Yaskawa INFORM job: SKRZYNIA_5540_0_STOPNI_1OBR.JBI

/JOB
//NAME SKRZYNIA_5540_0_STOPNI_1OBR
///FOLDERNAME 02-SKRZYNIE_JOBS
//POS
///NPOS 539,539,0,45,0,0
///TOOL 0
///POSTYPE PULSE
///PULSE
C00000=1055,-24125,84372,288,19725,204
C00001=1055,-24125,84372,288,19725,204
C00002=0,-15438,65714,0,-68532,0
C00003=25524,-25821,36823,19654,-58495,38520
C00004=25524,-25821,36823,19654,-58495,38520
C00005=23988,-24960,37134,18595,-57837,38812
C00006=22822,-23954,37534,17811,-57199,39017
C00007=22935,-24057,37491,17887,-57262,38997
C00008=20006,-24258,37408,15644,-56932,39751
C00009=24402,-25289,37013,18874,-58060,38740
C00010=22585,-24665,40358,17164,-59622,30036
C00011=23477,-23257,40205,18030,-58646,29630
C00012=22519,-22398,40568,17384,-58125,29795
C00013=22700,-22567,40495,17506,-58225,29764
C00014=19339,-22794,40398,14955,-57865,30607
C00015=24825,-24328,39798,18931,-59350,29401
C00016=25524,-25821,36823,19654,-58495,38520
C00017=23988,-24960,37134,18595,-57837,38812
C00018=22822,-23954,37534,17811,-57199,39017
C00019=22935,-24057,37491,17887,-57262,38997
C00020=20006,-24258,37408,15644,-56932,39751
C00021=24402,-25289,37013,18874,-58060,38740
C00022=22585,-24665,40358,17164,-59622,30036
C00023=23477,-23257,40205,18030,-58646,29630
C00024=22519,-22398,40568,17384,-58125,29795
C00025=22700,-22567,40495,17506,-58225,29764
C00026=19339,-22794,40398,14955,-57865,30607
C00027=24825,-24328,39798,18931,-59350,29401
C00028=32755,-32613,25711,29640,-48730,33694
C00029=25632,-30899,26166,23992,-46203,35378
C00030=24264,-29862,26497,22996,-45413,35639
C00031=24403,-29974,26459,23097,-45496,35612
C00032=20575,-30233,26374,19602,-44891,36810
C00033=26556,-31526,25988,24663,-46720,35206
C00034=30846,-32795,25752,28021,-48338,30427
C00035=24953,-30697,26306,23444,-45946,31743
C00036=23937,-29910,26558,22702,-45353,31936
C00037=24039,-29993,26530,22778,-45414,31916
C00038=20322,-30240,26449,19379,-44834,33080
C00039=25997,-31433,26093,24205,-46535,31545
C00040=26028,-43665,26580,-39946,8682,24640
C00041=27956,-30595,53065,-101898,6609,54413
C00042=26028,-43663,26580,-39944,8677,24639
C00043=38124,-35330,25507,26155,-45940,34419
C00044=17528,-33021,25719,14295,-44761,40001
C00045=28412,-21339,35361,20830,-70681,36412
C00046=27333,-20260,35973,20228,-70115,36596
C00047=27560,-20497,35837,20355,-70235,36556
C00048=24830,-20816,35654,18694,-69859,37222
C00049=28877,-18893,40191,20941,-72149,36569
C00050=27817,-32566,25782,25532,-47502,36865
C00051=25779,-31294,26110,24054,-46400,37243
C00052=24344,-30243,26427,23007,-45578,37515
C00053=24432,-30312,26405,23072,-45630,37498
C00054=20021,-30599,26315,19050,-44944,38872
C00055=26262,-31616,26021,24405,-46667,37153
C00056=27439,-32346,25835,25259,-47302,36935
C00057=26020,-31415,26075,24237,-46513,37193
C00058=24581,-30384,26384,23190,-45695,37464
C00059=24689,-30466,26358,23269,-45758,37444
C00060=20001,-30771,26264,18999,-45026,38899
C00061=26308,-31607,26026,24448,-46671,37139
C00062=27526,-32360,25834,25329,-47326,36914
C00063=24645,-40364,6410,30045,-34429,34156
C00064=22958,-37632,10123,27061,-35370,35326
C00065=22703,-41294,1722,31272,-29953,33282
C00066=19440,-41515,1663,27208,-29122,34832
C00067=25465,-43501,1200,33269,-31905,32752
C00068=54276,-43673,-470,62120,-47739,23626
C00069=54276,-43673,-470,62120,-47739,23626
C00070=41752,-40945,238,55421,-40682,25053
C00071=39867,-39951,547,54583,-39468,25162
C00072=39963,-40004,529,54625,-39531,25157
C00073=37168,-40414,400,52318,-38319,25966
C00074=43368,-42081,-2849,57747,-40820,23950
C00075=4794,-34097,38974,4189,-31824,-1302
C00076=4794,-34097,38974,4189,13412,-1302
C00077=11237,-37131,38982,-12694,5333,8253
///LIMIT ON
C00078=18252,-32243,53492,22663,-13662,-6677
///LIMIT OFF
C00079=13219,-33034,38361,14494,-24384,-4511
C00080=38095,-40136,7813,41252,-44156,24924
C00081=33231,-38681,8176,37792,-41757,25918
C00082=31538,-37640,8473,36716,-40716,26179
C00083=31687,-37737,8444,36811,-40809,26155
C00084=27389,-38154,8322,32773,-39589,27627
C00085=33834,-39023,8084,38175,-42120,25821
C00086=9520,-44470,15692,8941,-38846,5030
C00087=4264,-34194,25387,4006,-26954,-81856
C00088=17634,-23800,39238,9573,-31425,-73339
C00089=17634,-23800,39238,9573,-31425,-73339
C00090=16549,-22464,39800,8390,-30730,-72975
C00091=16684,-22641,39722,8536,-30818,-73021
C00092=16684,-19968,45512,8078,-32771,-72767
C00093=17634,-23800,39238,9573,-31425,-73339
C00094=17837,-21535,44509,9322,-33342,-73155
C00095=17837,-21535,44509,9322,-33342,-73155
C00096=16866,-20378,45014,8305,-32755,-72853
C00097=17032,-20588,44918,8481,-32857,-72905
C00098=17032,-17542,51480,8009,-35060,-72636
C00099=17837,-21535,44509,9322,-33342,-73155
C00100=-20829,-18800,50532,-12466,-37179,-77446
C00101=-19934,-17904,50946,-11618,-36715,-77676
C00102=-20044,-18019,50891,-11723,-36773,-77647
C00103=-20044,-15288,56753,-11218,-38713,-77950
C00104=-20966,-18928,50473,-12596,-37250,-77413
C00105=-20884,-26676,33664,-14451,-31668,-76336
C00106=-20884,-26676,33664,-14451,-31668,-76336
C00107=-19557,-25338,34176,-13080,-30873,-76751
C00108=-19691,-25483,34117,-13220,-30955,-76709
C00109=-19691,-22773,39998,-12506,-32911,-77106
C00110=-20642,-26447,33747,-14206,-31526,-76411
C00111=-33629,-40566,17444,-29603,-33447,-71192
C00112=-33629,-40566,17444,42578,-32312,-84654
C00113=-42160,-31266,16400,42578,-32312,-84654
C00114=-87798,-804,48829,-20188,-26072,-60966
C00115=-76454,-11934,10236,-25964,7954,-64922
C00116=-76448,-11928,10235,-25961,7944,-64914
C00117=-68643,-7759,-23318,-14097,50582,-74897
C00118=-70868,-8793,-8075,-29663,30364,-70765
C00119=-67243,-1968,12282,-49553,26687,-63567
C00120=-68655,-309,14069,-48513,25966,-64203
C00121=-67497,-1678,12591,-49367,26558,-63682
C00122=-71436,-723,2905,-26484,35140,-73726
C00123=-71436,176,6426,-27636,33595,-73066
C00124=-71434,778,8668,-28412,32633,-72624
C00125=-68624,-2689,-85,-28291,36551,-72622
C00126=-99375,3692,5712,40719,48607,-84097
C00127=-94964,4957,10918,40408,44640,-83792
C00128=-93063,6047,12199,39572,43744,-83178
C00129=-94964,4957,10918,40408,44640,-83792
C00130=-94964,5754,13918,41385,43553,-84439
C00131=-94964,4957,10918,40408,44640,-83792
C00132=-90271,-412,-5146,23417,46876,-76529
C00133=-83133,-4088,-8267,6704,41492,-71542
C00134=-83133,-4088,-8267,6704,41492,-71542
C00135=-83133,-4088,-8267,6704,41492,-11598
C00136=-83133,-16026,-8267,6704,41492,-11598
C00137=-83133,-16026,-8267,6704,41492,-11598
C00138=-48225,-19387,30619,3889,32460,-6728
C00139=56943,-39861,25115,1795,-37402,-69601
C00140=29960,-38386,-19607,-115769,-41858,-24264
C00141=65721,-6478,18155,-133323,-22195,3361
C00142=70544,4411,32968,-134868,-18623,4660
C00143=71874,8263,38598,-134556,-17327,4659
C00144=72629,9390,40002,-135279,-16924,5107
C00145=71441,7638,37831,-134139,-17555,4406
C00146=77146,8888,25050,-166574,-32612,18372
C00147=77146,10029,28643,-166204,-31014,18167
C00148=77146,11198,32202,-165803,-29459,17947
C00149=75508,4678,16951,-165715,-35157,17778
C00150=68680,12216,24468,-164340,-40455,-13359
C00151=68362,12845,25743,-164045,-40097,-13561
C00152=68362,13700,28585,-163752,-38808,-13742
C00153=68362,12845,25743,-164045,-40097,-13561
C00154=64993,-1168,28876,-102971,-10760,-49875
C00155=63888,481,30670,-102324,-11438,-50313
C00156=64993,-1168,28876,-102971,-10760,-49875
C00157=58588,-14653,4620,-120782,-19611,-35794
C00158=29960,-38386,-19607,-115769,-41858,-24264
C00159=56943,-39861,25115,1795,-37402,-69601
C00160=-1002,-39861,25115,1795,-37402,-69601
C00161=-1001,-39858,25114,1795,-37402,0
///LIMIT ON
C00162=6591,-33902,35532,5956,-1761,-1932
///LIMIT OFF
C00163=6592,-33900,35531,103508,-35512,-26314
C00164=-99253,-13690,44082,59847,13407,-31313
C00165=-85045,-36869,-4353,28502,-22832,-52282
C00166=-92346,-18713,13565,21110,-22545,-55257
C00167=-85370,-14218,16934,32905,-23649,-60330
C00168=-84150,-13282,17685,34842,-23935,-61163
C00169=-82877,-12536,18624,36445,-24482,-61818
C00170=-84150,-13282,17685,34842,-23935,-61163
C00171=-85467,-11480,19558,33086,-23405,-60436
C00172=-84150,-13282,17685,34842,-23935,-61163
C00173=-85732,-21202,11427,30682,-24763,-59235
C00174=-84559,-15616,15722,33768,-24118,-60665
C00175=-84150,-13282,17685,34842,-23935,-61163
C00176=-83260,-12880,18034,36130,-24218,-61709
C00177=-84150,-13282,17685,34842,-23935,-61163
C00178=-85365,-11775,19006,33430,-23307,-60600
C00179=-84150,-13282,17685,34842,-23935,-61163
C00180=-85786,-16909,14677,31743,-23900,-59790
C00181=-84150,-13282,17685,34842,-23935,-61163
C00182=-83215,-12861,18051,36194,-24233,-61735
C00183=-84150,-13282,17685,34842,-23935,-61163
C00184=-85327,-11825,18959,33476,-23327,-60618
C00185=-84150,-13282,17685,34842,-23935,-61163
C00186=-87841,-18519,13420,28367,-23534,-58339
C00187=-84150,-13282,17685,34842,-23935,-61163
C00188=-83292,-12894,18020,36083,-24208,-61688
C00189=-84150,-13282,17685,34842,-23935,-61163
C00190=-85185,-12008,18799,33646,-23400,-60687
C00191=-84150,-13282,17685,34842,-23935,-61163
C00192=-86371,-18277,13606,30568,-23951,-59265
C00193=-84345,-13370,17612,34554,-23873,-61041
C00194=-83240,-12871,18042,36158,-24225,-61720
C00195=-84345,-13370,17612,34554,-23873,-61041
C00196=-85365,-12110,18711,33368,-23345,-60568
C00197=-84345,-13370,17612,34554,-23873,-61041
C00198=-86191,-19647,12567,30467,-24278,-59187
C00199=-84345,-13372,17610,34552,-23873,-61039
C00200=-83096,-12807,18098,36363,-24268,-61804
C00201=-84345,-13372,17610,34552,-23873,-61039
C00202=-85268,-12232,18600,33480,-23393,-60612
C00203=-84345,-13372,17610,34552,-23873,-61039
C00204=-84814,-16043,15376,33312,-24093,-60464
C00205=-84104,-13265,17702,34906,-23948,-61189
C00206=-82960,-12743,18153,36555,-24313,-61887
C00207=-84104,-13265,17702,34906,-23948,-61189
C00208=-84979,-12194,18635,33901,-23496,-60788
C00209=-84104,-13265,17702,34906,-23948,-61189
C00210=-86610,-16845,14732,30573,-23614,-59301
C00211=-84104,-13265,17702,34906,-23948,-61189
C00212=-82793,-12667,18222,36790,-24370,-61986
C00213=-84104,-13265,17702,34906,-23948,-61189
C00214=-84888,-12305,18537,34004,-23540,-60830
C00215=-84104,-13265,17702,34906,-23948,-61189
C00216=-83806,-19585,12613,33764,-25080,-60559
C00217=-83675,-13072,17868,35530,-24083,-61453
C00218=-82553,-12556,18319,37130,-24451,-62127
C00219=-83675,-13072,17868,35530,-24083,-61453
C00220=-84378,-12223,18610,34735,-23716,-61138
C00221=-83675,-13072,17868,35530,-24083,-61453
C00222=-87149,-17993,13826,29513,-23647,-58830
C00223=-84104,-13265,17702,34906,-23948,-61189
C00224=-82640,-12594,18285,37014,-24425,-62079
C00225=-84104,-13265,17702,34906,-23948,-61189
C00226=-84792,-12429,18430,34119,-23592,-60877
C00227=-84104,-13265,17702,34906,-23948,-61189
C00228=-83583,-9185,30892,23668,-36042,-57025
C00229=-85789,-8328,35795,20592,-37093,-55378
C00230=-85786,-16735,14816,31782,-23869,-59812
C00231=-84103,-13263,17702,34906,-23947,-61191
C00232=-83225,-12865,18046,36177,-24227,-61729
C00233=-84103,-13263,17702,34906,-23947,-61191
C00234=-84774,-12447,18412,34138,-23599,-60886
C00235=-84103,-13263,17702,34906,-23947,-61191
C00236=-86149,-16246,6730,18897,-35239,-57128
C00237=-86244,-15289,7532,18875,-35060,-57127
C00238=-85361,-14893,7870,19824,-35193,-57574
C00239=-86244,-15289,7532,18875,-35060,-57127
C00240=-86889,-14409,8282,18264,-34784,-56850
C00241=-86244,-15289,7532,18875,-35060,-57127
C00242=-90262,-21765,2389,14114,-35574,-54847
C00243=-90262,-21765,2389,28730,-17672,-54847
C00244=-89967,-19086,25635,28730,-17672,-54847
C00245=568,-24029,84339,168,19981,112
C00246=568,-24677,83015,164,20405,113
C00247=101153,-24598,83176,165,20353,113
C00248=101153,-24598,83176,165,20353,113
C00249=89967,-19086,25635,-28730,-17672,54847
C00250=90262,-21765,2389,-28730,-17672,54847
C00251=86932,-18662,4771,-17876,-35519,56628
C00252=86578,-15436,7408,-18515,-35011,56957
C00253=85428,-14922,7844,-19753,-35183,57541
C00254=84405,-14447,8250,-20842,-35348,58054
C00255=85428,-14922,7844,-19753,-35183,57541
C00256=86134,-13973,8661,-19091,-34881,57237
C00257=85428,-14922,7844,-19753,-35183,57541
C00258=85786,-16735,14816,-31782,-23869,59812
C00259=83514,-12996,17929,-35760,-24132,61552
C00260=82296,-12429,18424,-37488,-24534,62281
C00261=83514,-12996,17929,-35760,-24132,61552
C00262=84266,-12085,18725,-34910,-23738,61214
C00263=83514,-12996,17929,-35760,-24132,61552
C00264=87323,-6914,39851,-18853,-38149,44508
C00265=83118,-12818,18089,-36330,-24263,61791
C00266=81969,-12276,18566,-37944,-24648,62472
C00267=83118,-12818,18089,-36330,-24263,61791
C00268=83927,-11846,18941,-35423,-23842,61433
C00269=83118,-12818,18089,-36330,-24263,61791
C00270=83806,-19585,12613,-33764,-25080,60559
C00271=83148,-12832,18077,-36287,-24254,61773
C00272=81889,-12236,18598,-38058,-24676,62520
C00273=83148,-12832,18077,-36287,-24254,61773
C00274=83900,-11930,18867,-35446,-23862,61440
C00275=83148,-12832,18077,-36287,-24254,61773
C00276=86610,-16845,14732,-30573,-23614,59301
C00277=82493,-13239,17725,-37070,-24559,62089
C00278=81442,-12739,18159,-38529,-24915,62703
C00279=82493,-13239,17725,-37070,-24559,62089
C00280=83435,-12133,18689,-36040,-24063,61682
C00281=82493,-13239,17725,-37070,-24559,62089
C00282=84814,-16043,15376,-33312,-24093,60464
C00283=82555,-13613,17404,-36910,-24580,62015
C00284=81369,-13053,17885,-38558,-24979,62709
C00285=82555,-13613,17404,-36910,-24580,62015
C00286=83568,-12431,18429,-35805,-24046,61580
C00287=82555,-13613,17404,-36910,-24580,62015
C00288=86191,-19647,12567,-30467,-24278,59187
C00289=82500,-13648,17375,-36975,-24607,62039
C00290=81594,-13224,17740,-38236,-24911,62571
C00291=82500,-13648,17375,-36975,-24607,62039
C00292=83449,-12543,18332,-35941,-24104,61633
C00293=82500,-13648,17375,-36975,-24607,62039
C00294=86371,-18277,13606,-30568,-23951,59265
C00295=82904,-13790,17251,-36416,-24470,61808
C00296=81796,-13275,17692,-37971,-24838,62464
C00297=82904,-13790,17251,-36416,-24470,61808
C00298=83696,-12867,18046,-35547,-24051,61466
C00299=82904,-13790,17251,-36416,-24470,61808
C00300=87841,-18519,13420,-28367,-23534,58339
C00301=82748,-13879,17174,-36603,-24542,61883
C00302=81789,-13434,17554,-37946,-24861,62449
C00303=82748,-13879,17174,-36603,-24542,61883
C00304=83603,-12888,18026,-35668,-24086,61514
C00305=82748,-13879,17174,-36603,-24542,61883
C00306=85786,-16909,14677,-31743,-23900,59790
C00307=82339,-14116,16972,-37087,-24733,62079
C00308=81557,-13752,17280,-38171,-24994,62536
C00309=82339,-14116,16972,-37087,-24733,62079
C00310=83390,-12909,18006,-35951,-24172,61633
C00311=82339,-14116,16972,-37087,-24733,62079
C00312=85732,-21202,11427,-30682,-24763,59235
C00313=82398,-14365,16763,-36952,-24745,62014
C00314=81340,-13876,17176,-38416,-25096,62632
C00315=82398,-14365,16763,-36952,-24745,62014
C00316=83629,-12951,17972,-35620,-24090,61491
C00317=82398,-14365,16763,-36952,-24745,62014
C00318=92346,-18713,13565,-21110,-22545,55257
C00319=82794,-13980,17083,-36511,-24538,61844
C00320=81697,-13472,17516,-38043,-24902,62488
C00321=82794,-13980,17083,-36511,-24538,61844
C00322=83767,-12847,18056,-35444,-24023,61424
C00323=82794,-13980,17083,-36511,-24538,61844
C00324=85045,-36869,-4353,-28502,-22832,52282
C00325=69856,-53931,-13446,-33557,-28911,29591
C00326=0,-24029,84339,0,19981,0
C00327=0,-24029,84339,0,19981,0
C00328=0,-52280,40443,0,6876,0
C00329=43695,-41610,22646,45477,-37580,9181
C00330=79833,-32060,29151,65065,-75499,17030
C00331=46589,-23543,32575,47437,-59456,19719
C00332=21464,-32103,9331,16221,-60878,34097
C00333=58029,-25484,23838,55879,-68285,17494
C00334=64424,-28491,31029,58630,-66351,17656
C00335=0,-52280,40443,0,6876,0
C00336=0,-52280,40443,0,6876,0
C00337=23755,-47704,18289,26329,-25233,13971
C00338=32804,-46073,6525,41905,-31120,14425
C00339=62562,-39100,6547,70046,-55853,12125
C00340=48126,-33841,8393,64372,-47199,12361
C00341=14189,-48092,-16375,12117,-40492,32069
C00342=59828,-44646,-5405,72855,-48572,12139
///LIMIT ON
C00343=0,-38761,66314,0,-763,0
C00344=0,-44757,54667,0,2744,0
///LIMIT OFF
C00345=40382,-38226,12225,48505,-40693,16039
C00346=55481,-27484,23768,62968,-54833,11978
C00347=49599,-26598,24185,59764,-51822,12602
C00348=49350,-31368,12250,54913,-55857,13157
C00349=55330,-33748,11238,57660,-59334,12681
C00350=78664,-24436,10378,82837,-79111,12029
C00351=75189,-23065,11287,81851,-76948,11927
C00352=75189,-45249,11287,81851,-38847,11927
C00353=29880,-45249,11287,43145,-11324,11927
C00354=0,-24029,84339,0,19981,0
C00355=0,-24026,84338,1,19977,2
C00356=4264,-34194,25387,4006,-26954,-29436
C00357=4264,-34194,25387,4006,-26954,-81856
C00358=-21478,-27798,32214,-15234,-31599,-76056
C00359=-19679,-23059,39354,-12567,-32689,-77067
C00360=16724,-20576,44291,8212,-32395,-72836
C00361=21329,-26386,39716,13285,-34016,-74401
C00362=-23778,-26243,38799,-16502,-35132,-75964
C00363=-20075,-15782,55752,-11329,-38404,-77896
C00364=16874,-17447,51356,7863,-34895,-72604
C00365=18580,-28601,30698,11472,-29284,-74138
C00366=-2794,-29341,30774,-2918,-30250,-75106
C00367=-922,-23070,40815,-1467,-32356,-75153
C00368=2749,-22947,41081,710,-32295,-74788
C00369=21329,-26386,39716,13285,-34016,-74401
C00370=6126,-41331,18955,6697,-26557,-30383
C00371=1,-24024,84337,2,19973,1
C00372=-64243,-26178,31107,-39513,40312,-5844
C00373=-72148,3973,56008,-35470,42045,-10522
C00374=-72090,16396,76301,-42067,35650,-6519
C00375=-69388,15725,61378,-31740,35177,-8719
C00376=-69127,27099,75569,-32744,34250,-8088
C00377=-67573,2495,11285,-21767,57629,-15193
C00378=-77819,19629,29798,-10454,63174,-20704
C00379=-72990,23583,14304,-10735,77209,-20379
C00380=-74593,38003,46707,-11043,65751,-19814
C00381=-73236,38943,48295,-11400,65557,-19316
C00382=-73329,42107,51779,-6346,67443,-19636
C00383=-87142,34654,46174,17622,63862,-25393
C00384=-87240,36727,48611,18897,66604,-25032
C00385=-99033,21517,12213,24947,79702,-26203
C00386=-91500,-14196,-34781,24472,81625,-22832
C00387=-100472,-45007,-27818,8167,67201,-29302
C00388=0,-36642,16905,0,48372,0
C00389=66009,-61997,-62105,21406,63483,18379
C00390=97242,-23579,-39442,10179,68876,30321
C00391=73684,-7073,-17511,24638,68131,29022
C00392=59136,7235,6676,33270,66602,27507
C00393=54816,14937,6234,39741,69494,31070
C00394=54365,20668,19279,41017,66202,29418
C00395=64503,4223,2857,29650,48528,26647
C00396=75622,3202,-3149,3890,49494,34281
C00397=88036,13177,2413,-18568,66573,35876
C00398=90462,21593,10123,-22613,76266,34479
C00399=92450,29224,20002,-25750,81642,33727
C00400=94949,8131,-12163,-20291,74229,36861
C00401=94949,8084,-13484,-20215,75047,36712
C00402=70412,-34016,-52305,-11724,65624,29757
C00403=44268,-30306,-1568,-7370,48673,18708
C00404=1,-24024,84337,2,19973,1
C00405=1,-24024,84337,2,19973,1
C00406=3796,-57671,22373,2336,-25309,-753
C00407=52632,-34554,16626,51161,-63050,5622
C00408=59461,-32779,9832,66317,-58406,17312
C00409=52597,-27799,19145,60250,-56477,14854
C00410=30424,-23087,38603,28410,-55402,26626
C00411=62932,-33588,12189,66848,-61063,18031
C00412=55769,-31640,17107,64026,-54372,11197
C00413=49589,-26873,23592,59558,-52024,12630
C00414=49411,-31351,12257,54953,-55883,13142
C00415=55330,-33748,11238,57660,-59334,12681
C00416=62932,-33588,12189,66848,-61063,18031
C00417=1,-24024,84337,2,19973,1
C00418=1,-24024,84337,2,19973,1
C00419=57188,-41777,19973,48132,-58706,4905
C00420=55566,-48748,-16991,79805,-45048,-6941
C00421=49908,-48716,-25784,90749,-41340,-3650
C00422=43952,-47082,-25409,90867,-37558,-4523
C00423=43999,-46718,-25278,91104,-37601,-4657
C00424=55479,-50244,-26473,91085,-44870,-3042
///LIMIT ON
C00425=12119,-24859,71505,13236,4440,2633
///LIMIT OFF
C00426=-91085,-34291,10385,1908,-24348,-42097
C00427=-86191,-19647,12567,30467,-24278,-59187
C00428=-99148,-11667,19101,-13975,-20192,-40187
C00429=-98206,-11518,19604,-10142,-20308,-41629
C00430=-99474,-20389,12397,-11593,-22150,-41069
C00431=0,-52280,40443,0,6876,0
C00432=98750,-34911,19055,13387,-20552,33529
C00433=85481,-22689,10385,-30594,-25183,59147
C00434=96971,-12584,18294,8365,-19955,42614
C00435=97182,-12918,18001,8747,-20027,42449
C00436=96230,-24528,9149,6144,-22576,43630
C00437=0,-52280,40443,0,6876,0
C00438=0,-52280,40443,0,6876,0
///LIMIT ON
C00439=-90140,-60305,18108,-2708,1721,-7625
///LIMIT OFF
C00440=-95594,-27428,6866,-4663,-19832,-42154
C00441=-99356,-13410,18355,-15385,-17730,-37479
C00442=-99405,-10878,20508,-15853,-17333,-37255
C00443=-99132,-10804,20575,-15274,-17279,-37502
C00444=-99172,-3396,39216,-11005,-24351,-39647
C00445=-98898,-3229,39076,-10663,-24101,-39776
C00446=-100183,-18601,14070,-16273,-18800,-37146
///LIMIT ON
C00447=-90140,-60305,18108,-2708,1721,-7625
///LIMIT OFF
C00448=0,-52280,40443,0,6876,0
///LIMIT ON
C00449=84259,-57935,27522,-3761,3673,6310
///LIMIT OFF
C00450=86507,-39672,4297,-27618,-16640,46340
C00451=79502,-31038,5321,-35142,-29552,60614
C00452=87509,-17632,14108,-29072,-23467,58651
C00453=100395,-12639,18246,19464,-20904,37830
C00454=99174,-17330,4434,32315,-9754,28887
C00455=99172,-17333,4433,32310,-9754,28889
C00456=98988,-17100,4624,31837,-9651,29097
C00457=100388,-17987,13832,15751,-21517,39479
C00458=86507,-39672,4297,-27618,-16640,46340
///LIMIT ON
C00459=84259,-57935,27522,-3761,3673,6310
///LIMIT OFF
C00460=0,-52280,40443,0,6876,0
C00461=0,-27933,77061,0,20812,0
C00462=0,-27933,77061,0,20812,0
C00463=0,-52280,40443,0,6876,0
///LIMIT ON
C00464=-91970,-60791,14435,-3343,512,-9412
///LIMIT OFF
C00465=-99196,-15868,16098,-13748,-19297,-38710
C00466=-99196,-15868,16098,-13748,-19297,-38710
C00467=-99196,-15868,16098,-13748,-19297,-38710
C00468=-85815,-11758,19597,31748,-21097,-58265
C00469=-87383,-11883,19487,26986,-20206,-56250
C00470=-99562,-16264,15781,-14410,-19427,-38431
C00471=-99196,-15868,16098,-13748,-19297,-38710
///LIMIT ON
C00472=-91970,-60791,14435,-3343,512,-9412
///LIMIT OFF
C00473=0,-52280,40443,0,6876,0
///LIMIT ON
C00474=91083,-60784,14823,-9043,-825,15173
///LIMIT OFF
C00475=83869,-19403,12921,-33769,-24740,60260
C00476=83869,-19403,12921,-33769,-24740,60260
C00477=83420,-14897,16486,-35538,-24144,61113
C00478=90567,-11796,19696,-13982,-20789,51525
C00479=90367,-11588,19943,-14262,-20865,51612
C00480=95871,-14889,15992,4901,-19605,43825
C00481=83869,-19403,12921,-33769,-24740,60260
///LIMIT ON
C00482=91083,-60784,14823,-9043,-825,15173
///LIMIT OFF
C00483=0,-52280,40443,0,6876,0
///LIMIT ON
C00484=-91526,-60598,16699,7584,176,-13289
///LIMIT OFF
C00485=-94392,-6553,48683,5805,-47321,-49764
C00486=-88951,-345,54953,10686,-47392,-51569
C00487=-88172,5833,62122,11322,-47753,-51785
C00488=-90949,-14015,9500,8834,-34399,-51934
C00489=-84917,-15593,15742,33275,-23984,-60461
C00490=-81669,-15982,15425,37506,-25258,-62202
C00491=-79867,-25377,9541,37586,-25936,-59971
///LIMIT ON
C00492=-91415,-60262,16631,7870,-73,-13734
///LIMIT OFF
C00493=24,-24029,84339,7,19981,5
C00494=160,-24029,84339,47,19981,32
C00495=99096,-24029,84339,47,19981,32
C00496=99096,-24029,84339,47,19981,32
C00497=89967,-19086,25635,-28730,-17672,54847
C00498=85786,-16735,14816,-31782,-23869,59812
C00499=83492,-14473,16674,-35480,-24338,61406
C00500=82709,-11470,19305,-37370,-24374,62232
C00501=85293,-13629,8874,-19696,-34851,57583
C00502=85505,-16299,6686,-19564,-35388,57437
C00503=89967,-19086,25635,-28730,-17672,54847
C00504=568,-24029,84339,168,19981,112
C00505=568,-24029,84339,168,19981,112
///LIMIT ON
C00506=-91970,-60791,14435,-3343,512,-9412
///LIMIT OFF
C00507=-86948,-23217,10819,28314,-23349,-56438
C00508=-85895,-16522,15767,31843,-22281,-58087
C00509=-93643,1708,52973,2937,-38210,-34777
C00510=-93409,-737,47229,3345,-36106,-34967
C00511=-86145,-24679,9854,29028,-23971,-56682
///LIMIT ON
C00512=-100471,-58311,4157,14142,-4822,-27614
C00513=-68517,-58311,4157,14142,-4822,-27614
///LIMIT OFF
C00514=0,-52280,40443,0,6876,0
///LIMIT ON
C00515=91083,-60784,14823,-9043,-825,15173
///LIMIT OFF
C00516=83869,-19403,12921,-33769,-24740,60260
C00517=82620,-18743,14708,-32942,-26226,58979
C00518=83315,-11405,20766,-33572,-24860,59408
C00519=83357,-11106,21030,-33564,-24812,59409
C00520=84798,-22668,11879,-29033,-26372,57255
///LIMIT ON
C00521=91083,-60784,14823,-9043,-825,15173
///LIMIT OFF
C00522=0,-52280,40443,0,6876,0
///LIMIT ON
C00523=-6369,-39206,65423,-4801,-482,2563
///LIMIT OFF
C00524=-97287,-29142,12714,-8673,-22288,-37832
C00525=-86191,-19647,12567,30467,-24278,-59187
C00526=-85671,-16302,15857,30808,-24404,-58999
C00527=-99988,-10363,22448,-14642,-22536,-38816
C00528=-95800,-10799,21862,-1195,-21693,-44692
C00529=-87910,-17792,15835,25414,-24996,-56048
C00530=-97287,-29142,12714,-8673,-22288,-37832
C00531=0,-52280,40443,0,6876,0
C00532=92301,-25634,22749,2368,-15645,37646
C00533=83738,-18329,13570,-34202,-24868,60772
C00534=90157,-13013,18222,-15321,-20860,52657
C00535=93373,-13178,17985,-4546,-20133,48070
C00536=80226,-20465,12178,-39626,-27411,62762
C00537=92301,-25634,22749,2368,-15645,37646
C00538=0,-52280,40443,0,6876,0
BC00000=428499
BC00001=428499
BC00002=428499
BC00003=428495
BC00004=305607
BC00005=305607
BC00006=305607
BC00007=305607
BC00008=305607
BC00009=305607
BC00010=362488
BC00011=362493
BC00012=362493
BC00013=362493
BC00014=362493
BC00015=362493
BC00016=428495
BC00017=428495
BC00018=428495
BC00019=428495
BC00020=428495
BC00021=428495
BC00022=489984
BC00023=489989
BC00024=489989
BC00025=489989
BC00026=489989
BC00027=489989
BC00028=538210
BC00029=538210
BC00030=538210
BC00031=538210
BC00032=538210
BC00033=538210
BC00034=601406
BC00035=601406
BC00036=601406
BC00037=601406
BC00038=601406
BC00039=601406
BC00040=494983
BC00041=634221
BC00042=689318
BC00043=706706
BC00044=702330
BC00045=727611
BC00046=727611
BC00047=727611
BC00048=727611
BC00049=727611
BC00050=723631
BC00051=723631
BC00052=723631
BC00053=723631
BC00054=723631
BC00055=723631
BC00056=785545
BC00057=785545
BC00058=785545
BC00059=785545
BC00060=785545
BC00061=785545
BC00062=839091
BC00063=845328
BC00064=845330
BC00065=845331
BC00066=845331
BC00067=845331
BC00068=848702
BC00069=906836
BC00070=906836
BC00071=906836
BC00072=906836
BC00073=906836
BC00074=906836
BC00075=755710
BC00076=703061
BC00077=787304
BC00078=898647
BC00079=924265
BC00080=965197
BC00081=965197
BC00082=965197
BC00083=965197
BC00084=965197
BC00085=965197
BC00086=954305
BC00087=972596
BC00088=987957
BC00089=987957
BC00090=987957
BC00091=987957
BC00092=987957
BC00093=987957
BC00094=992403
BC00095=992403
BC00096=992403
BC00097=992403
BC00098=992403
BC00099=992403
BC00100=992403
BC00101=992403
BC00102=992403
BC00103=992403
BC00104=992403
BC00105=992403
BC00106=992403
BC00107=992403
BC00108=992403
BC00109=992403
BC00110=992403
BC00111=992403
BC00112=992403
BC00113=992403
BC00114=992403
BC00115=992403
BC00116=1010155
BC00117=1021241
BC00118=1037945
BC00119=1037945
BC00120=1037945
BC00121=1037945
BC00122=1037945
BC00123=1037945
BC00124=1037946
BC00125=1037946
BC00126=1037946
BC00127=1037946
BC00128=1037946
BC00129=1037946
BC00130=1037946
BC00131=1037946
BC00132=1028323
BC00133=1013689
BC00134=988424
BC00135=988424
BC00136=988424
BC00137=955242
BC00138=920809
BC00139=992403
BC00140=992403
BC00141=992403
BC00142=1008617
BC00143=1013778
BC00144=1013778
BC00145=1013778
BC00146=1013778
BC00147=1013778
BC00148=1013778
BC00149=1013778
BC00150=1013778
BC00151=1013778
BC00152=1013778
BC00153=1013778
BC00154=1013778
BC00155=1013778
BC00156=1013778
BC00157=1008265
BC00158=961681
BC00159=930959
BC00160=930959
BC00161=946322
BC00162=877259
BC00163=877262
BC00164=877262
BC00165=946865
BC00166=978995
BC00167=978992
BC00168=978992
BC00169=978992
BC00170=978992
BC00171=978992
BC00172=978992
BC00173=917549
BC00174=917549
BC00175=917549
BC00176=917549
BC00177=917549
BC00178=917549
BC00179=917549
BC00180=856105
BC00181=856105
BC00182=856105
BC00183=856105
BC00184=856105
BC00185=856105
BC00186=794661
BC00187=794661
BC00188=794661
BC00189=794661
BC00190=794661
BC00191=794661
BC00192=733216
BC00193=733216
BC00194=733216
BC00195=733216
BC00196=733216
BC00197=733216
BC00198=671766
BC00199=671766
BC00200=671766
BC00201=671766
BC00202=671766
BC00203=671766
BC00204=610322
BC00205=610322
BC00206=610322
BC00207=610322
BC00208=610322
BC00209=610322
BC00210=548878
BC00211=548878
BC00212=548878
BC00213=548878
BC00214=548878
BC00215=548878
BC00216=487434
BC00217=487434
BC00218=487434
BC00219=487434
BC00220=487434
BC00221=487434
BC00222=425990
BC00223=425990
BC00224=425990
BC00225=425990
BC00226=425990
BC00227=425990
BC00228=425990
BC00229=364547
BC00230=364547
BC00231=364547
BC00232=364547
BC00233=364547
BC00234=364547
BC00235=364547
BC00236=351830
BC00237=351830
BC00238=351830
BC00239=351830
BC00240=351830
BC00241=351830
BC00242=351830
BC00243=351830
BC00244=351830
BC00245=351830
BC00246=526918
BC00247=527366
BC00248=379158
BC00249=351830
BC00250=351830
BC00251=352776
BC00252=352776
BC00253=352776
BC00254=352776
BC00255=352776
BC00256=352776
BC00257=352776
BC00258=364547
BC00259=365498
BC00260=365498
BC00261=365498
BC00262=365498
BC00263=365498
BC00264=425990
BC00265=426941
BC00266=426941
BC00267=426941
BC00268=426941
BC00269=426941
BC00270=487434
BC00271=488386
BC00272=488386
BC00273=488386
BC00274=488386
BC00275=488386
BC00276=548878
BC00277=549829
BC00278=549829
BC00279=549829
BC00280=549829
BC00281=549829
BC00282=610322
BC00283=610322
BC00284=610322
BC00285=610322
BC00286=610322
BC00287=610322
BC00288=671766
BC00289=672711
BC00290=672711
BC00291=672711
BC00292=672711
BC00293=672711
BC00294=733216
BC00295=734160
BC00296=734160
BC00297=734160
BC00298=734160
BC00299=734160
BC00300=794661
BC00301=795606
BC00302=795606
BC00303=795606
BC00304=795606
BC00305=795606
BC00306=856105
BC00307=857052
BC00308=857052
BC00309=857052
BC00310=857052
BC00311=857052
BC00312=917549
BC00313=918497
BC00314=918497
BC00315=918497
BC00316=918497
BC00317=918497
BC00318=978995
BC00319=978994
BC00320=978994
BC00321=978994
BC00322=978994
BC00323=978994
BC00324=946865
BC00325=825529
BC00326=750988
BC00327=785327
BC00328=732226
BC00329=738956
BC00330=732532
BC00331=732532
BC00332=731145
BC00333=731361
BC00334=742986
BC00335=732226
BC00336=873772
BC00337=936552
BC00338=962717
BC00339=971247
BC00340=970959
BC00341=970959
BC00342=961243
BC00343=855481
BC00344=554334
BC00345=500587
BC00346=472057
BC00347=472057
BC00348=432637
BC00349=432637
BC00350=509347
BC00351=529667
BC00352=529667
BC00353=529667
BC00354=509347
BC00355=866230
BC00356=954347
BC00357=959563
BC00358=992403
BC00359=992403
BC00360=987956
BC00361=982190
BC00362=977701
BC00363=992403
BC00364=992403
BC00365=991631
BC00366=992045
BC00367=990150
BC00368=989717
BC00369=982190
BC00370=995223
BC00371=843084
BC00372=858446
BC00373=858446
BC00374=915156
BC00375=935042
BC00376=959981
BC00377=991913
BC00378=991913
BC00379=1019422
BC00380=1019422
BC00381=1019422
BC00382=1019423
BC00383=1019423
BC00384=1019424
BC00385=1019424
BC00386=1019424
BC00387=934082
BC00388=892680
BC00389=976220
BC00390=1015340
BC00391=1015341
BC00392=1015341
BC00393=1045588
BC00394=1045588
BC00395=1045588
BC00396=1045588
BC00397=1045588
BC00398=1045591
BC00399=1045591
BC00400=1045591
BC00401=1019185
BC00402=1019185
BC00403=950372
BC00404=827723
BC00405=492012
BC00406=537922
BC00407=581892
BC00408=609309
BC00409=609309
BC00410=545209
BC00411=545209
BC00412=349169
BC00413=347429
BC00414=310527
BC00415=309749
BC00416=545209
BC00417=476651
BC00418=678676
BC00419=793675
BC00420=793673
BC00421=793673
BC00422=793673
BC00423=853583
BC00424=853583
BC00425=581771
BC00426=722718
BC00427=671766
BC00428=671766
BC00429=733216
BC00430=733216
BC00431=733216
BC00432=677664
BC00433=672711
BC00434=672711
BC00435=734164
BC00436=734164
BC00437=733216
BC00438=808033
BC00439=808033
BC00440=912211
BC00441=911081
BC00442=911081
BC00443=972539
BC00444=972539
BC00445=993822
BC00446=972539
BC00447=808033
BC00448=808033
BC00449=808033
BC00450=902807
BC00451=918487
BC00452=918487
BC00453=918487
BC00454=979938
BC00455=991458
BC00456=1009173
BC00457=979938
BC00458=902807
BC00459=808033
BC00460=808033
BC00461=715610
BC00462=561575
BC00463=561575
BC00464=561572
BC00465=561572
BC00466=422137
BC00467=422137
BC00468=422139
BC00469=483561
BC00470=483561
BC00471=561572
BC00472=561572
BC00473=561575
BC00474=561575
BC00475=522965
BC00476=426143
BC00477=426143
BC00478=426143
BC00479=488081
BC00480=488081
BC00481=522965
BC00482=561575
BC00483=561575
BC00484=532118
BC00485=399077
BC00486=364547
BC00487=364547
BC00488=351830
BC00489=364547
BC00490=425990
BC00491=431873
BC00492=531162
BC00493=535379
BC00494=489374
BC00495=489374
BC00496=418469
BC00497=351830
BC00498=364547
BC00499=364547
BC00500=364547
BC00501=352776
BC00502=352776
BC00503=351830
BC00504=351830
BC00505=443762
BC00506=561572
BC00507=606449
BC00508=606449
BC00509=606449
BC00510=546477
BC00511=545001
BC00512=545001
BC00513=545001
BC00514=545001
BC00515=561575
BC00516=605280
BC00517=610988
BC00518=610988
BC00519=549538
BC00520=549538
BC00521=561575
BC00522=545001
BC00523=666556
BC00524=781251
BC00525=793329
BC00526=793814
BC00527=794613
BC00528=856109
BC00529=856109
BC00530=781251
BC00531=733216
BC00532=756461
BC00533=795585
BC00534=795583
BC00535=857104
BC00536=857104
BC00537=756461
BC00538=733216
///POSTYPE BASE
///RECTAN
///RCONF 1,0,0,0,0,0,0,0,0,0,0,0,0,0,0,0,0,0,0,0,0,0,0,0
P00006=0.000,0.000,0.000,0.0000,0.0000,0.0000
///RCONF 0,0,0,0,0,0,0,0,0,0,0,0,0,0,0,0,0,0,0,0,0,0,0,0
P00021=6.550,-0.003,-5.735,0.0000,0.0000,0.0000
P00022=5.943,-0.018,-6.388,0.0000,0.0000,0.0000
P00023=7.025,-0.019,-7.168,0.0000,0.0000,0.0000
P00024=5.926,-0.047,-4.777,0.0000,0.0000,0.0000
///RCONF 1,0,0,0,0,0,0,0,0,0,0,0,0,0,0,0,0,0,0,0,0,0,0,0
P00098=-0.089,-2.467,4.059,0.0000,0.0000,0.0000
P00099=0.011,-2.380,1.226,0.0000,0.0000,0.0000
P00100=-0.081,2.558,4.482,0.0000,0.0000,0.0000
P00101=0.030,-2.286,2.993,0.0000,0.0000,0.0000
P00102=-0.005,-1.108,1.644,0.0000,0.0000,0.0000
P00103=-0.094,-3.400,4.200,0.0000,0.0000,0.0000
P00104=0.043,-2.127,5.826,0.0000,0.0000,0.0000
P00105=-0.043,0.662,5.286,0.0000,0.0000,0.0000
P00106=-0.018,-2.519,0.237,0.0000,0.0000,0.0000
P00107=-0.008,-4.537,-4.500,0.0000,0.0000,0.0000
P00108=0.014,-3.040,2.637,0.0000,0.0000,0.0000
P00109=0.017,-3.622,2.341,0.0000,0.0000,0.0000
///RCONF 0,0,0,0,0,0,0,0,0,0,0,0,0,0,0,0,0,0,0,0,0,0,0,0
P00280=-0.761,-1.221,0.004,0.0000,0.0000,0.0000
///RCONF 1,0,0,0,0,0,0,0,0,0,0,0,0,0,0,0,0,0,0,0,0,0,0,0
P00281=-0.866,-3.587,-0.008,0.0000,0.0000,0.0000
///RCONF 0,0,0,0,1,0,0,0,0,0,0,0,0,0,0,0,0,0,0,0,0,0,0,0
P00290=-0.023,-0.050,5.560,0.0000,0.0000,0.0000
///RCONF 1,0,0,0,0,0,0,0,0,0,0,0,0,0,0,0,0,0,0,0,0,0,0,0
P00291=0.002,-0.893,4.526,0.0000,0.0000,0.0000
P00300=-0.036,-1.505,2.318,0.0000,0.0000,0.0000
P00301=0.046,-2.112,7.779,0.0000,0.0000,0.0000
P00302=-0.180,-2.409,6.326,0.0000,0.0000,0.0000
///RCONF 0,0,0,0,0,0,0,0,0,0,0,0,0,0,0,0,0,0,0,0,0,0,0,0
P00303=-0.004,-1.437,-4.584,0.0000,0.0000,0.0000
P00304=0.028,-1.666,-4.234,0.0000,0.0000,0.0000
P00305=-0.003,-1.920,-3.501,0.0000,0.0000,0.0000
P00306=0.015,-2.252,-3.054,0.0000,0.0000,0.0000
P00307=0.019,-2.151,-5.077,0.0000,0.0000,0.0000
P00308=-0.003,-2.092,-4.888,0.0000,0.0000,0.0000
P00309=-0.040,-2.205,-4.992,0.0000,0.0000,0.0000
P00310=-0.006,-2.490,-5.925,0.0000,0.0000,0.0000
P00311=-0.007,-2.079,-5.307,0.0000,0.0000,0.0000
P00350=11.519,-0.008,1.149,0.0000,0.0000,0.0000
P00351=13.563,-0.027,-0.653,0.0000,0.0000,0.0000
P00352=13.252,-0.027,-0.827,0.0000,0.0000,0.0000
P00353=10.971,-0.082,0.776,0.0000,0.0000,0.0000
P00354=-0.024,2.508,-1.824,0.0000,0.0000,0.0000
P00355=-0.001,2.528,-1.131,0.0000,0.0000,0.0000
P00356=-0.034,2.921,-0.262,0.0000,0.0000,0.0000
P00357=0.003,3.386,-0.091,0.0000,0.0000,0.0000
P00358=0.014,3.037,-0.020,0.0000,0.0000,0.0000
P00359=-0.005,2.731,0.912,0.0000,0.0000,0.0000
P00360=-0.011,3.412,0.438,0.0000,0.0000,0.0000
P00361=0.018,3.050,1.253,0.0000,0.0000,0.0000
//INST
///DATE 2025/02/20 14:15
///ATTR SC,RW
///GROUP1 RB1,BS1
NOP
CALL JOB:MOVE_INTO_TUNNEL
MOVJ C00000 BC00000 VJ=30.00
'------------------------
'------------------------
'SPOINA SRODEK DOL
'------------------------
'------------------------
'POMIAR DO WYJ!! PRZEROBIC NA STD
MOVJ C00001 BC00001 VJ=40.00
MOVJ C00002 BC00002 VJ=40.00
'W3P
MOVJ C00003 BC00003 VJ=20.00 PL=0
'SPOINA_PODLOGA_BRAK_ROZP
MOVJ C00004 BC00004 VJ=20.00 PL=0
MOVL C00005 BC00005 V=166.7 PL=0
REFP 3 C00006 BC00006
CALL JOB:SEARCH-R1
SET P0098 P0006
SFTON P0098
MOVL C00007 BC00007 V=66.7 PL=0
REFP 3 C00008 BC00008
CALL JOB:SEARCH-R1
SET P0098 P0006
SFTON P0098
MOVL C00009 BC00009 V=333.3 PL=0
SFTOF
'W3L
MOVL C00010 BC00010 V=666.7
MOVL C00011 BC00011 V=166.7 PL=0
REFP 3 C00012 BC00012
CALL JOB:SEARCH-R1
SET P0099 P0006
SFTON P0099
MOVL C00013 BC00013 V=166.7 PL=0
REFP 3 C00014 BC00014
CALL JOB:SEARCH-R1
SET P0099 P0006
SFTON P0099
MOVL C00015 BC00015 V=333.3 PL=0
SFTOF
'SPOINA_PODLOGA_BRAK_ROZP
MOVJ C00016 BC00016 VJ=20.00 PL=0
MOVL C00017 BC00017 V=166.7 PL=0
REFP 3 C00018 BC00018
CALL JOB:SEARCH-R1
SET P0100 P0006
SFTON P0100
MOVL C00019 BC00019 V=66.7 PL=0
REFP 3 C00020 BC00020
CALL JOB:SEARCH-R1
SET P0100 P0006
SFTON P0100
MOVL C00021 BC00021 V=333.3 PL=0
SFTOF
'W3L
MOVL C00022 BC00022 V=666.7
MOVL C00023 BC00023 V=166.7 PL=0
REFP 3 C00024 BC00024
CALL JOB:SEARCH-R1
SET P0101 P0006
SFTON P0101
MOVL C00025 BC00025 V=166.7 PL=0
REFP 3 C00026 BC00026
CALL JOB:SEARCH-R1
SET P0101 P0006
SFTON P0101
MOVL C00027 BC00027 V=333.3 PL=0
SFTOF
'W9P
MOVL C00028 BC00028 V=666.7
MOVL C00029 BC00029 V=166.7
REFP 3 C00030 BC00030
CALL JOB:SEARCH-R1
SET P0102 P0006
SFTON P0102
MOVL C00031 BC00031 V=166.7 PL=0
REFP 3 C00032 BC00032
CALL JOB:SEARCH-R1
SET P0102 P0006
SFTON P0102
MOVL C00033 BC00033 V=333.3 PL=0
'W9L
MOVL C00034 BC00034 V=666.7
MOVL C00035 BC00035 V=166.7
REFP 3 C00036 BC00036
CALL JOB:SEARCH-R1
SET P0103 P0006
SFTON P0103
MOVL C00037 BC00037 V=166.7 PL=0
REFP 3 C00038 BC00038
CALL JOB:SEARCH-R1
SET P0103 P0006
SFTON P0103
MOVL C00039 BC00039 V=333.3 PL=0
SFTOF
'PRZEJAZ NAD BELKA
MOVL C00040 BC00040 V=666.7
MOVJ C00041 BC00041 VJ=40.00
MOVJ C00042 BC00042 VJ=40.00
MOVJ C00043 BC00043 VJ=40.00
'W1P
SFTOF
MOVJ C00044 BC00044 VJ=20.00 PL=0
MOVL C00045 BC00045 V=166.7 PL=0
REFP 3 C00046 BC00046
CALL JOB:SEARCH-R1
SET P0104 P0006
SFTON P0104
MOVL C00047 BC00047 V=166.7 PL=0
REFP 3 C00048 BC00048
CALL JOB:SEARCH-R1
SET P0104 P0006
SFTON P0104
MOVL C00049 BC00049 V=333.3 PL=0
SFTOF
'W1L
MOVL C00050 BC00050 V=666.7
MOVL C00051 BC00051 V=166.7 PL=0
REFP 3 C00052 BC00052
CALL JOB:SEARCH-R1
SET P0105 P0006
SFTON P0105
MOVL C00053 BC00053 V=166.7 PL=0
REFP 3 C00054 BC00054
CALL JOB:SEARCH-R1
SET P0105 P0006
SFTON P0105
MOVL C00055 BC00055 V=333.3 PL=0
SFTOF
MOVL C00056 BC00056 V=666.7
'W10P
MOVL C00057 BC00057 V=166.7 PL=0
REFP 3 C00058 BC00058
CALL JOB:SEARCH-R1
SET P0106 P0006
SFTON P0106
MOVL C00059 BC00059 V=166.7 PL=0
REFP 3 C00060 BC00060
CALL JOB:SEARCH-R1
SET P0106 P0006
SFTON P0106
MOVL C00061 BC00061 V=333.3 PL=0
SFTOF
'W10L
MOVL C00062 BC00062 V=333.3
MOVL C00063 BC00063 V=166.7 PL=0
REFP 3 C00064 BC00064
CALL JOB:SEARCH-R1
SET P0107 P0006
SFTON P0107
MOVL C00065 BC00065 V=166.7 PL=0
REFP 3 C00066 BC00066
CALL JOB:SEARCH-R1
SET P0107 P0006
SFTON P0107
MOVL C00067 BC00067 V=333.3 PL=0
SFTOF
MOVL C00068 BC00068 V=333.3
MOVL C00069 BC00069 V=333.3
MOVL C00070 BC00070 V=166.7 PL=0
REFP 3 C00071 BC00071
CALL JOB:SEARCH-R1
SET P0108 P0006
SFTON P0108
MOVL C00072 BC00072 V=166.7 PL=0
REFP 3 C00073 BC00073
CALL JOB:SEARCH-R1
SET P0108 P0006
SFTON P0108
MOVL C00074 BC00074 V=333.3 PL=0
SFTOF
'PRZEJAZD
MOVJ C00075 BC00075 VJ=50.00
MOVJ C00076 BC00076 VJ=50.00
MOVJ C00077 BC00077 VJ=60.00
MOVJ C00078 BC00078 VJ=60.00
MOVJ C00079 BC00079 VJ=60.00
'W2P
'W2L
MOVL C00080 BC00080 V=666.7
MOVL C00081 BC00081 V=166.7 PL=0
REFP 3 C00082 BC00082
CALL JOB:SEARCH-R1
SET P0109 P0006
SFTON P0109
MOVL C00083 BC00083 V=166.7 PL=0
REFP 3 C00084 BC00084
CALL JOB:SEARCH-R1
SET P0109 P0006
SFTON P0109
MOVL C00085 BC00085 V=333.3 PL=0
SFTOF
MOVJ C00086 BC00086 VJ=40.00
MOVJ C00087 BC00087 VJ=50.00
'W5L
MOVJ C00088 BC00088 VJ=30.00 PL=0
MOVL C00089 BC00089 V=166.7
REFP 3 C00090 BC00090
CALL JOB:SEARCH-R1
SET P0021 P0006
SFTON P0021
MOVL C00091 BC00091 V=166.7
REFP 3 C00092 BC00092
CALL JOB:SEARCH-R1
SET P0021 P0006
SFTON P0021
SFTOF
MOVL C00093 BC00093 V=166.7
'W6L
MOVJ C00094 BC00094 VJ=20.00 PL=0
MOVL C00095 BC00095 V=166.7
REFP 3 C00096 BC00096
CALL JOB:SEARCH-R1
SET P0022 P0006
SFTON P0022
MOVL C00097 BC00097 V=166.7
REFP 3 C00098 BC00098
CALL JOB:SEARCH-R1
SET P0022 P0006
SFTON P0022
SFTOF
MOVL C00099 BC00099 V=166.7
'W6P
MOVL C00100 BC00100 V=333.3 PL=0
REFP 3 C00101 BC00101
CALL JOB:SEARCH-R1
SET P0023 P0006
SFTON P0023
MOVL C00102 BC00102 V=166.7
REFP 3 C00103 BC00103
CALL JOB:SEARCH-R1
SET P0023 P0006
SFTON P0023
SFTOF
MOVL C00104 BC00104 V=166.7
'W5P
MOVJ C00105 BC00105 VJ=20.00 PL=0
MOVL C00106 BC00106 V=166.7
REFP 3 C00107 BC00107
CALL JOB:SEARCH-R1
SET P0024 P0006
SFTON P0024
MOVL C00108 BC00108 V=166.7
REFP 3 C00109 BC00109
CALL JOB:SEARCH-R1
SET P0024 P0006
SFTON P0024
SFTOF
MOVL C00110 BC00110 V=166.7
'W7A
MOVJ C00111 BC00111 VJ=40.00
MOVJ C00112 BC00112 VJ=40.00
MOVJ C00113 BC00113 VJ=40.00
MOVJ C00114 BC00114 VJ=40.00
MOVJ C00115 BC00115 VJ=40.00
MOVJ C00116 BC00116 VJ=40.00
MOVJ C00117 BC00117 VJ=40.00
MOVJ C00118 BC00118 VJ=40.00
MOVL C00119 BC00119 V=250.0
REFP 3 C00120 BC00120
CALL JOB:SEARCH-R1
SET P0280 P0006
SFTON P0280
MOVL C00121 BC00121 V=166.7
MOVL C00122 BC00122 V=250.0
MOVL C00123 BC00123 V=166.7
REFP 3 C00124 BC00124
CALL JOB:SEARCH-R1
SET P0280 P0006
MOVL C00125 BC00125 V=166.7
SFTOF
MOVL C00126 BC00126 V=333.3
MOVL C00127 BC00127 V=166.7
REFP 3 C00128 BC00128
CALL JOB:SEARCH-R1
SET P0290 P0006
SFTON P0290
MOVL C00129 BC00129 V=166.7
REFP 3 C00130 BC00130
CALL JOB:SEARCH-R1
SET P0290 P0006
MOVL C00131 BC00131 V=166.7
MOVJ C00132 BC00132 VJ=20.00
SFTOF
MOVJ C00133 BC00133 VJ=30.00
MOVJ C00134 BC00134 VJ=40.00
MOVJ C00135 BC00135 VJ=40.00
MOVJ C00136 BC00136 VJ=40.00
MOVJ C00137 BC00137 VJ=40.00
MOVJ C00138 BC00138 VJ=50.00
'W7B
MOVJ C00139 BC00139 VJ=50.00
MOVJ C00140 BC00140 VJ=50.00
MOVJ C00141 BC00141 VJ=30.00
MOVJ C00142 BC00142 VJ=20.00
MOVL C00143 BC00143 V=166.7
REFP 3 C00144 BC00144
CALL JOB:SEARCH-R1
SET P0281 P0006
MOVL C00145 BC00145 V=166.7
SFTON P0281
MOVL C00146 BC00146 V=166.7
MOVL C00147 BC00147 V=166.7
REFP 3 C00148 BC00148
CALL JOB:SEARCH-R1
SET P0281 P0006
MOVJ C00149 BC00149 VJ=15.00
SFTOF
MOVJ C00150 BC00150 VJ=20.00
MOVL C00151 BC00151 V=166.7
REFP 3 C00152 BC00152
CALL JOB:SEARCH-R1
SET P0291 P0006
MOVL C00153 BC00153 V=166.7
MOVL C00154 BC00154 V=166.7
REFP 3 C00155 BC00155
CALL JOB:SEARCH-R1
SET P0291 P0006
MOVL C00156 BC00156 V=166.7
MOVJ C00157 BC00157 VJ=30.00
MOVJ C00158 BC00158 VJ=30.00
MOVJ C00159 BC00159 VJ=50.00
MOVJ C00160 BC00160 VJ=50.00
'------------------------
'------------------------
'PRAWA STRONA PROFIL GORA
'------------------------
'------------------------
MOVJ C00161 BC00161 VJ=50.00
MOVJ C00162 BC00162 VJ=50.00
MOVJ C00163 BC00163 VJ=50.00
MOVJ C00164 BC00164 VJ=20.00
MOVJ C00165 BC00165 VJ=50.00
'------------------------
'W14A L
'------------------------
SFTOF
MOVJ C00166 BC00166 VJ=50.00
MOVJ C00167 BC00167 VJ=30.00
MOVL C00168 BC00168 V=166.7 PL=0
REFP 3 C00169 BC00169
CALL JOB:SEARCH-R1
SET P0300 P0006
SFTON P0300
MOVL C00170 BC00170 V=166.7 PL=0
REFP 3 C00171 BC00171
CALL JOB:SEARCH-R1
SET P0300 P0006
SFTON P0300
MOVL C00172 BC00172 V=166.7 PL=0
SFTOF
'------------------------
'W14A P
'------------------------
SFTOF
MOVJ C00173 BC00173 VJ=50.00
MOVJ C00174 BC00174 VJ=50.00
MOVL C00175 BC00175 V=166.7 PL=0
REFP 3 C00176 BC00176
CALL JOB:SEARCH-R1
SET P0301 P0006
SFTON P0301
MOVL C00177 BC00177 V=166.7 PL=0
REFP 3 C00178 BC00178
CALL JOB:SEARCH-R1
SET P0301 P0006
SFTON P0301
MOVL C00179 BC00179 V=166.7 PL=0
SFTOF
'------------------------
'W19A L
'------------------------
SFTOF
MOVJ C00180 BC00180 VJ=50.00
MOVL C00181 BC00181 V=200.0 PL=0
REFP 3 C00182 BC00182
CALL JOB:SEARCH-R1
SET P0302 P0006
SFTON P0302
MOVL C00183 BC00183 V=166.7 PL=0
REFP 3 C00184 BC00184
CALL JOB:SEARCH-R1
SET P0302 P0006
SFTON P0302
MOVL C00185 BC00185 V=250.0 PL=0
SFTOF
'------------------------
'W19A P
'------------------------
SFTOF
MOVJ C00186 BC00186 VJ=50.00
MOVL C00187 BC00187 V=166.7 PL=0
REFP 3 C00188 BC00188
CALL JOB:SEARCH-R1
SET P0303 P0006
SFTON P0303
MOVL C00189 BC00189 V=166.7 PL=0
REFP 3 C00190 BC00190
CALL JOB:SEARCH-R1
SET P0303 P0006
SFTON P0303
MOVL C00191 BC00191 V=166.7 PL=0
SFTOF
'------------------------
'W13A L
'------------------------
SFTOF
MOVJ C00192 BC00192 VJ=50.00
MOVL C00193 BC00193 V=166.7 PL=0
REFP 3 C00194 BC00194
CALL JOB:SEARCH-R1
SET P0304 P0006
SFTON P0304
MOVL C00195 BC00195 V=166.7 PL=0
REFP 3 C00196 BC00196
CALL JOB:SEARCH-R1
SET P0304 P0006
SFTON P0304
MOVL C00197 BC00197 V=166.7 PL=0
SFTOF
'------------------------
'W13A P
'------------------------
SFTOF
MOVJ C00198 BC00198 VJ=50.00
MOVL C00199 BC00199 V=200.0 PL=0
REFP 3 C00200 BC00200
CALL JOB:SEARCH-R1
SET P0305 P0006
SFTON P0305
MOVL C00201 BC00201 V=166.7 PL=0
REFP 3 C00202 BC00202
CALL JOB:SEARCH-R1
SET P0305 P0006
SFTON P0305
MOVL C00203 BC00203 V=250.0 PL=0
SFTOF
'------------------------
'W18A L
'------------------------
SFTOF
MOVJ C00204 BC00204 VJ=50.00
MOVL C00205 BC00205 V=200.0 PL=0
REFP 3 C00206 BC00206
CALL JOB:SEARCH-R1
SET P0306 P0006
SFTON P0306
MOVL C00207 BC00207 V=166.7 PL=0
REFP 3 C00208 BC00208
CALL JOB:SEARCH-R1
SET P0306 P0006
SFTON P0306
MOVL C00209 BC00209 V=166.7 PL=0
SFTOF
'------------------------
'W18A P
'------------------------
SFTOF
MOVJ C00210 BC00210 VJ=50.00
MOVL C00211 BC00211 V=200.0 PL=0
REFP 3 C00212 BC00212
CALL JOB:SEARCH-R1
SET P0307 P0006
SFTON P0307
MOVL C00213 BC00213 V=166.7 PL=0
REFP 3 C00214 BC00214
CALL JOB:SEARCH-R1
SET P0307 P0006
SFTON P0307
MOVL C00215 BC00215 V=166.7 PL=0
SFTOF
'------------------------
'W15A L
'------------------------
SFTOF
MOVJ C00216 BC00216 VJ=50.00
MOVL C00217 BC00217 V=200.0 PL=0
REFP 3 C00218 BC00218
CALL JOB:SEARCH-R1
SET P0308 P0006
SFTON P0308
MOVL C00219 BC00219 V=166.7 PL=0
REFP 3 C00220 BC00220
CALL JOB:SEARCH-R1
SET P0308 P0006
SFTON P0308
MOVL C00221 BC00221 V=166.7 PL=0
SFTOF
'------------------------
'W15A P
'------------------------
SFTOF
MOVJ C00222 BC00222 VJ=50.00
MOVL C00223 BC00223 V=166.7 PL=0
REFP 3 C00224 BC00224
CALL JOB:SEARCH-R1
SET P0309 P0006
SFTON P0309
MOVL C00225 BC00225 V=166.7 PL=0
REFP 3 C00226 BC00226
CALL JOB:SEARCH-R1
SET P0309 P0006
SFTON P0309
MOVL C00227 BC00227 V=166.7 PL=0
SFTOF
MOVL C00228 BC00228 V=333.3
'------------------------
'W17A L
'------------------------
MOVL C00229 BC00229 V=500.0
SFTOF
MOVJ C00230 BC00230 VJ=20.00
MOVL C00231 BC00231 V=166.7 PL=0
REFP 3 C00232 BC00232
CALL JOB:SEARCH-R1
SET P0310 P0006
SFTON P0310
MOVL C00233 BC00233 V=166.7 PL=0
REFP 3 C00234 BC00234
CALL JOB:SEARCH-R1
SET P0310 P0006
SFTON P0310
MOVL C00235 BC00235 V=166.7 PL=0
SFTOF
'------------------------
'W17A P
'------------------------
SFTOF
MOVL C00236 BC00236 V=416.7
MOVL C00237 BC00237 V=166.7 PL=0
REFP 3 C00238 BC00238
CALL JOB:SEARCH-R1
SET P0311 P0006
SFTON P0311
MOVL C00239 BC00239 V=166.7 PL=0
REFP 3 C00240 BC00240
CALL JOB:SEARCH-R1
SET P0311 P0006
SFTON P0311
MOVL C00241 BC00241 V=166.7 PL=0
SFTOF
MOVJ C00242 BC00242 VJ=10.00
MOVJ C00243 BC00243 VJ=20.00
MOVJ C00244 BC00244 VJ=50.00
MOVJ C00245 BC00245 VJ=50.00
MOVJ C00246 BC00246 VJ=70.00
MOVJ C00247 BC00247 VJ=30.00
MOVJ C00248 BC00248 VJ=30.00
'------------------------
'------------------------
'LEWA STRONA PROFIL GORA
'------------------------
'------------------------
MOVJ C00249 BC00249 VJ=30.00
MOVJ C00250 BC00250 VJ=30.00
MOVJ C00251 BC00251 VJ=30.00
'------------------------
'W17B L
'------------------------
SFTOF
MOVJ C00252 BC00252 VJ=15.00
MOVL C00253 BC00253 V=166.7 PL=0
REFP 3 C00254 BC00254
CALL JOB:SEARCH-R1
SET P0350 P0006
SFTON P0350
MOVL C00255 BC00255 V=166.7 PL=0
REFP 3 C00256 BC00256
CALL JOB:SEARCH-R1
SET P0350 P0006
SFTON P0350
MOVL C00257 BC00257 V=166.7 PL=0
SFTOF
'------------------------
'W17B P
'------------------------
SFTOF
MOVL C00258 BC00258 V=333.3
MOVL C00259 BC00259 V=166.7 PL=0
REFP 3 C00260 BC00260
CALL JOB:SEARCH-R1
SET P0351 P0006
SFTON P0351
MOVL C00261 BC00261 V=166.7 PL=0
REFP 3 C00262 BC00262
CALL JOB:SEARCH-R1
SET P0351 P0006
SFTON P0351
MOVL C00263 BC00263 V=166.7 PL=0
SFTOF
'POPRAWID DOJAZD
'------------------------
'W15B L
'------------------------
SFTOF
MOVJ C00264 BC00264 VJ=10.00
MOVL C00265 BC00265 V=166.7 PL=0
REFP 3 C00266 BC00266
CALL JOB:SEARCH-R1
SET P0352 P0006
SFTON P0352
MOVL C00267 BC00267 V=166.7 PL=0
REFP 3 C00268 BC00268
CALL JOB:SEARCH-R1
SET P0352 P0006
SFTON P0352
MOVL C00269 BC00269 V=166.7 PL=0
SFTOF
'------------------------
'W15B P
'------------------------
SFTOF
MOVJ C00270 BC00270 VJ=20.00
MOVL C00271 BC00271 V=166.7 PL=0
REFP 3 C00272 BC00272
CALL JOB:SEARCH-R1
SET P0353 P0006
SFTON P0353
MOVL C00273 BC00273 V=166.7 PL=0
REFP 3 C00274 BC00274
CALL JOB:SEARCH-R1
SET P0353 P0006
SFTON P0353
MOVL C00275 BC00275 V=166.7 PL=0
SFTOF
'------------------------
'W18B L
'------------------------
SFTOF
MOVJ C00276 BC00276 VJ=50.00
MOVL C00277 BC00277 V=166.7 PL=0
REFP 3 C00278 BC00278
CALL JOB:SEARCH-R1
SET P0354 P0006
SFTON P0354
MOVL C00279 BC00279 V=166.7 PL=0
REFP 3 C00280 BC00280
CALL JOB:SEARCH-R1
SET P0354 P0006
SFTON P0354
MOVL C00281 BC00281 V=166.7 PL=0
SFTOF
'------------------------
'W18B P
'------------------------
SFTOF
MOVJ C00282 BC00282 VJ=50.00
MOVL C00283 BC00283 V=166.7 PL=0
REFP 3 C00284 BC00284
CALL JOB:SEARCH-R1
SET P0355 P0006
SFTON P0355
MOVL C00285 BC00285 V=166.7 PL=0
REFP 3 C00286 BC00286
CALL JOB:SEARCH-R1
SET P0355 P0006
SFTON P0355
MOVL C00287 BC00287 V=166.7 PL=0
SFTOF
'------------------------
'W13B L
'------------------------
SFTOF
MOVJ C00288 BC00288 VJ=50.00
MOVL C00289 BC00289 V=166.7 PL=0
REFP 3 C00290 BC00290
CALL JOB:SEARCH-R1
SET P0356 P0006
SFTON P0356
MOVL C00291 BC00291 V=166.7 PL=0
REFP 3 C00292 BC00292
CALL JOB:SEARCH-R1
SET P0356 P0006
SFTON P0356
MOVL C00293 BC00293 V=166.7 PL=0
SFTOF
'------------------------
'W13B P
'------------------------
SFTOF
MOVJ C00294 BC00294 VJ=50.00
MOVL C00295 BC00295 V=166.7 PL=0
REFP 3 C00296 BC00296
CALL JOB:SEARCH-R1
SET P0357 P0006
SFTON P0357
MOVL C00297 BC00297 V=166.7 PL=0
REFP 3 C00298 BC00298
CALL JOB:SEARCH-R1
SET P0357 P0006
SFTON P0357
MOVL C00299 BC00299 V=166.7 PL=0
SFTOF
'------------------------
'W19B L
'------------------------
SFTOF
MOVJ C00300 BC00300 VJ=50.00
MOVL C00301 BC00301 V=166.7 PL=0
REFP 3 C00302 BC00302
CALL JOB:SEARCH-R1
SET P0358 P0006
SFTON P0358
MOVL C00303 BC00303 V=166.7 PL=0
REFP 3 C00304 BC00304
CALL JOB:SEARCH-R1
SET P0358 P0006
SFTON P0358
MOVL C00305 BC00305 V=166.7 PL=0
SFTOF
'------------------------
'W19B P
'------------------------
SFTOF
MOVJ C00306 BC00306 VJ=50.00
MOVL C00307 BC00307 V=166.7 PL=0
REFP 3 C00308 BC00308
CALL JOB:SEARCH-R1
SET P0359 P0006
SFTON P0359
MOVL C00309 BC00309 V=166.7 PL=0
REFP 3 C00310 BC00310
CALL JOB:SEARCH-R1
SET P0359 P0006
SFTON P0359
MOVL C00311 BC00311 V=166.7 PL=0
SFTOF
'------------------------
'W14B L
'------------------------
SFTOF
MOVJ C00312 BC00312 VJ=50.00
MOVL C00313 BC00313 V=166.7 PL=0
REFP 3 C00314 BC00314
CALL JOB:SEARCH-R1
SET P0360 P0006
SFTON P0360
MOVL C00315 BC00315 V=166.7 PL=0
REFP 3 C00316 BC00316
CALL JOB:SEARCH-R1
SET P0360 P0006
SFTON P0360
MOVL C00317 BC00317 V=166.7 PL=0
SFTOF
'------------------------
'W14B P
'------------------------
SFTOF
MOVJ C00318 BC00318 VJ=50.00
MOVL C00319 BC00319 V=166.7 PL=0
REFP 3 C00320 BC00320
CALL JOB:SEARCH-R1
SET P0361 P0006
SFTON P0361
MOVL C00321 BC00321 V=166.7 PL=0
REFP 3 C00322 BC00322
CALL JOB:SEARCH-R1
SET P0361 P0006
SFTON P0361
MOVL C00323 BC00323 V=166.7 PL=0
SFTOF
MOVJ C00324 BC00324 VJ=50.00
MOVJ C00325 BC00325 VJ=50.00
MOVJ C00326 BC00326 VJ=50.00
'WELD
'WELD
'WELD
MOVJ C00327 BC00327 VJ=10.00
'**********************
'**********************
'POCZATEK SPAWANIA DOL
'**********************
'**********************
''
'**********************
'W1
'**********************
MOVJ C00328 BC00328 VJ=50.00
MOVJ C00329 BC00329 VJ=40.00
MOVL C00330 BC00330 V=166.7
SFTON P0105
MOVL C00331 BC00331 V=166.7
MACRO1 MJ#(0) ARGF24
ARCON
SFTON P0104
MOVL C00332 BC00332 V=11.3
ARCOF
SFTOF
MOVL C00333 BC00333 V=333.3
MOVJ C00334 BC00334 VJ=20.00
MOVJ C00335 BC00335 VJ=30.00
MOVJ C00336 BC00336 VJ=50.00
MOVJ C00337 BC00337 VJ=40.00
MOVJ C00338 BC00338 VJ=20.00
'**********************
'W2
'**********************
MOVL C00339 BC00339 V=166.7
SFTON P0109
MOVL C00340 BC00340 V=333.3
ARCON
SFTON P0108
MOVL C00341 BC00341 V=10.8
ARCOF
SFTOF
MOVL C00342 BC00342 V=333.3
MOVJ C00343 BC00343 VJ=40.00
MOVJ C00344 BC00344 VJ=70.00
MOVJ C00345 BC00345 VJ=20.00
MOVL C00346 BC00346 V=666.7
'**********************
'W3
'**********************
SFTON P0101
MOVL C00347 BC00347 V=166.7
ARCON
SFTON P0100
MOVL C00348 BC00348 V=11.7
ARCOF
MOVL C00349 BC00349 V=166.7
SFTOF
MOVJ C00350 BC00350 VJ=30.00
MOVJ C00351 BC00351 VJ=30.00
MOVJ C00352 BC00352 VJ=50.00
MOVJ C00353 BC00353 VJ=30.00
MOVJ C00354 BC00354 VJ=40.00
'**********************
'W5
'**********************
MOVJ C00355 BC00355 VJ=50.00
MOVJ C00356 BC00356 VJ=25.00
MOVJ C00357 BC00357 VJ=30.00
'**********************
'W5
MOVL C00358 BC00358 V=333.3
'**********************
MACRO1 MJ#(0) ARGF9
SFTON P0024
MOVL C00359 BC00359 V=166.7
ARCON
WVON WEV#(2)
SFTON P0021
MOVL C00360 BC00360 V=10.8
ARCOF
WVOF
SFTOF
MOVJ C00361 BC00361 VJ=20.00
MOVJ C00362 BC00362 VJ=20.00
'**********************
'W6
'**********************
MACRO1 MJ#(0) ARGF9
SFTON P0023
MOVL C00363 BC00363 V=250.0
ARCON
WVON WEV#(2)
SFTON P0022
MOVL C00364 BC00364 V=10.8
ARCOF
WVOF
SFTOF
MOVJ C00365 BC00365 VJ=10.00
MOVL C00366 BC00366 V=333.3
'**********************
MACRO1 MJ#(0) ARGF9
SFTON P0024
MOVL C00367 BC00367 V=166.7
ARCON
WVON WEV#(3)
SFTON P0021
MOVL C00368 BC00368 V=10.8
ARCOF
WVOF
SFTOF
MOVJ C00369 BC00369 VJ=20.00
MOVJ C00370 BC00370 VJ=30.00
MOVJ C00371 BC00371 VJ=40.00
MOVJ C00372 BC00372 VJ=40.00
MOVJ C00373 BC00373 VJ=40.00
MOVJ C00374 BC00374 VJ=40.00
MOVJ C00375 BC00375 VJ=20.00
MOVJ C00376 BC00376 VJ=10.00
MOVJ C00377 BC00377 VJ=20.00
MOVL C00378 BC00378 V=166.7
MACRO1 MJ#(0) ARGF14
MOVL C00379 BC00379 V=166.7
SFTON P0280
MOVL C00380 BC00380 V=166.7 PL=0
ARCON ASF#(22)
MOVL C00381 BC00381 V=9.2
MOVL C00382 BC00382 V=9.2
SFTON P0281
MOVL C00383 BC00383 V=9.2
MOVL C00384 BC00384 V=9.2
ARCOF
SFTOF
MOVL C00385 BC00385 V=250.0
MOVL C00386 BC00386 V=416.7
MOVJ C00387 BC00387 VJ=30.00
MOVJ C00388 BC00388 VJ=30.00
MOVJ C00389 BC00389 VJ=30.00
MOVJ C00390 BC00390 VJ=30.00
MOVJ C00391 BC00391 VJ=30.00
'7b
MOVL C00392 BC00392 V=333.3
MOVL C00393 BC00393 V=333.3
SFTON P0281
MOVL C00394 BC00394 V=166.7 PL=0
ARCON ASF#(22)
MOVL C00395 BC00395 V=9.2
MOVL C00396 BC00396 V=9.2
SFTON P0291
MOVL C00397 BC00397 V=9.2
MOVL C00398 BC00398 V=9.2
MOVL C00399 BC00399 V=9.2
ARCOF
SFTOF
'TUTAJ DODAC 7
'TUTAJ DODAC 7
'TUTAJ DODAC 7
MOVL C00400 BC00400 V=333.3
MOVL C00401 BC00401 V=333.3
MOVL C00402 BC00402 V=333.3
MOVJ C00403 BC00403 VJ=20.00
MOVJ C00404 BC00404 VJ=30.00
MOVJ C00405 BC00405 VJ=50.00
MOVJ C00406 BC00406 VJ=50.00
MOVJ C00407 BC00407 VJ=40.00
MOVJ C00408 BC00408 VJ=10.00
'**********************
'W9
'**********************
SFTON P0103
MACRO1 MJ#(0) ARGF24
MOVL C00409 BC00409 V=166.7
ARCON
SFTON P0102
MOVL C00410 BC00410 V=11.3
ARCOF
SFTOF
MOVL C00411 BC00411 V=166.7
'**********************
'SPOINA_PODLOGA_BRAK_ROZP
'**********************
MOVL C00412 BC00412 V=333.3
SFTON P0099
MOVL C00413 BC00413 V=166.7
ARCON
SFTON P0098
MOVL C00414 BC00414 V=11.7
ARCOF
MOVL C00415 BC00415 V=166.7
SFTOF
'SPOINA_PODLOGA_BRAK_ROZP
MOVL C00416 BC00416 V=166.7
MOVJ C00417 BC00417 VJ=40.00
MOVJ C00418 BC00418 VJ=70.00
MOVJ C00419 BC00419 VJ=50.00
MOVJ C00420 BC00420 VJ=20.00
'**********************
'W10
'**********************
MOVL C00421 BC00421 V=333.3
SFTON P0106
MOVL C00422 BC00422 V=166.7
ARCON
SFTON P0107
MOVL C00423 BC00423 V=11.3
ARCOF
SFTOF
MOVL C00424 BC00424 V=333.3
MOVJ C00425 BC00425 VJ=50.00
'**********************
'**********************
'POCZATEK SPAWANIA BOKI
'**********************
'**********************
MOVJ C00426 BC00426 VJ=50.00
MOVJ C00427 BC00427 VJ=50.00
'**********************
'W13A
'**********************
SFTON P0305
MOVL C00428 BC00428 V=250.0 PL=0
SFTOF
MACRO1 MJ#(0) ARGF10
ARCON
SFTON P0304
MOVL C00429 BC00429 V=10.8
ARCOF
SFTOF
MOVL C00430 BC00430 V=250.0
'W13B
MOVJ C00431 BC00431 VJ=30.00
MOVJ C00432 BC00432 VJ=50.00
MOVL C00433 BC00433 V=500.0
'**********************
'W13B
'**********************
SFTON P0356
MOVL C00434 BC00434 V=16.7 PL=0
SFTOF
ARCON
SFTON P0357
MOVL C00435 BC00435 V=10.8
ARCOF
SFTOF
MOVL C00436 BC00436 V=250.0
MOVJ C00437 BC00437 VJ=30.00
MOVJ C00438 BC00438 VJ=40.00
MOVJ C00439 BC00439 VJ=30.00
MOVJ C00440 BC00440 VJ=30.00
'**********************
'W14A
'**********************
MOVL C00441 BC00441 V=250.0
SFTON P0301
MOVL C00442 BC00442 V=50.0 PL=0
SFTOF
ARCON
SFTON P0300
MOVL C00443 BC00443 V=10.8
MOVL C00444 BC00444 V=10.8
MOVL C00445 BC00445 V=10.8
ARCOF
SFTOF
MOVL C00446 BC00446 V=150.0
MOVJ C00447 BC00447 VJ=40.00
MOVJ C00448 BC00448 VJ=30.00
MOVJ C00449 BC00449 VJ=30.00
MOVJ C00450 BC00450 VJ=30.00
MOVJ C00451 BC00451 VJ=30.00
'**********************
'W14B
'**********************
SFTON P0360
MOVL C00452 BC00452 V=333.3
MOVL C00453 BC00453 V=166.7 PL=0
SFTOF
ARCON
SFTON P0361
MOVL C00454 BC00454 V=10.8
MOVL C00455 BC00455 V=10.8
MOVL C00456 BC00456 V=10.8
ARCOF
SFTOF
MOVL C00457 BC00457 V=250.0
MOVJ C00458 BC00458 VJ=40.00
MOVJ C00459 BC00459 VJ=40.00
MOVJ C00460 BC00460 VJ=30.00
MOVJ C00461 BC00461 VJ=40.00
MOVJ C00462 BC00462 VJ=30.00
MOVJ C00463 BC00463 VJ=30.00
MOVJ C00464 BC00464 VJ=30.00
MOVJ C00465 BC00465 VJ=30.00
MOVJ C00466 BC00466 VJ=30.00
'**********************
'W15A
'**********************
SFTON P0309
MOVL C00467 BC00467 V=166.7
MOVL C00468 BC00468 V=166.7 PL=0
SFTOF
ARCON
SFTON P0308
MOVL C00469 BC00469 V=10.8
ARCOF
SFTOF
MOVL C00470 BC00470 V=150.0
MOVJ C00471 BC00471 VJ=30.00
MOVJ C00472 BC00472 VJ=50.00
MOVJ C00473 BC00473 VJ=50.00
MOVJ C00474 BC00474 VJ=50.00
MOVJ C00475 BC00475 VJ=50.00
MOVJ C00476 BC00476 VJ=50.00
'**********************
'W15B
'**********************
SFTON P0352
MOVL C00477 BC00477 V=250.0
MOVL C00478 BC00478 V=83.3 PL=0
SFTOF
ARCON
SFTON P0353
MOVL C00479 BC00479 V=10.8
ARCOF
MOVL C00480 BC00480 V=66.7
SFTOF
MOVJ C00481 BC00481 VJ=40.00
MOVJ C00482 BC00482 VJ=50.00
MOVJ C00483 BC00483 VJ=50.00
'BRAK W TEJ DLUGOSCI
'**********************
'W16A
'**********************
'**********************
'W16B
'**********************
'BRAK W TEJ DLUGOSCI
'**********************
'W17A
'**********************
MOVJ C00484 BC00484 VJ=50.00
MOVJ C00485 BC00485 VJ=50.00
'**********************
'W17A
'**********************
SFTON P0310
MOVL C00486 BC00486 V=333.3
MOVL C00487 BC00487 V=166.7 PL=0
SFTOF
ARCON
SFTON P0311
MOVL C00488 BC00488 V=10.8
ARCOF
SFTOF
MOVL C00489 BC00489 V=333.3
MOVJ C00490 BC00490 VJ=30.00
MOVJ C00491 BC00491 VJ=30.00
MOVJ C00492 BC00492 VJ=50.00
MOVJ C00493 BC00493 VJ=50.00
MOVJ C00494 BC00494 VJ=50.00
MOVJ C00495 BC00495 VJ=50.00
MOVJ C00496 BC00496 VJ=50.00
MOVJ C00497 BC00497 VJ=30.00
MOVJ C00498 BC00498 VJ=30.00
'**********************
'W17B
'**********************
SFTON P0351
MOVL C00499 BC00499 V=166.7
MOVL C00500 BC00500 V=166.7 PL=0
SFTOF
ARCON
SFTON P0350
MOVL C00501 BC00501 V=10.8
ARCOF
SFTOF
MOVL C00502 BC00502 V=250.0
MOVJ C00503 BC00503 VJ=30.00
MOVJ C00504 BC00504 VJ=30.00
MOVJ C00505 BC00505 VJ=30.00
MOVJ C00506 BC00506 VJ=30.00
MOVJ C00507 BC00507 VJ=40.00
'**********************
'W18A
'**********************
SFTON P0306
MOVL C00508 BC00508 V=333.3
MOVL C00509 BC00509 V=166.7 PL=0
SFTOF
ARCON
SFTON P0307
MOVL C00510 BC00510 V=10.8
ARCOF
SFTOF
MOVL C00511 BC00511 V=250.0
MOVJ C00512 BC00512 VJ=30.00
MOVJ C00513 BC00513 VJ=30.00
MOVJ C00514 BC00514 VJ=50.00
MOVJ C00515 BC00515 VJ=50.00
MOVJ C00516 BC00516 VJ=50.00
'**********************
'W18B
'**********************
SFTON P0355
MOVL C00517 BC00517 V=166.7
MOVL C00518 BC00518 V=166.7 PL=0
SFTOF
ARCON
SFTON P0354
MOVL C00519 BC00519 V=10.8
ARCOF
MOVL C00520 BC00520 V=250.0
SFTOF
MOVJ C00521 BC00521 VJ=30.00
MOVJ C00522 BC00522 VJ=30.00
MOVJ C00523 BC00523 VJ=40.00
MOVJ C00524 BC00524 VJ=50.00
MOVJ C00525 BC00525 VJ=30.00
'**********************
'W19A
'**********************
MOVL C00526 BC00526 V=166.7
SFTON P0303
MOVL C00527 BC00527 V=166.7 PL=0
SFTOF
ARCON
SFTON P0302
MOVL C00528 BC00528 V=10.8
ARCOF
SFTOF
MOVL C00529 BC00529 V=150.0
MOVJ C00530 BC00530 VJ=30.00
MOVJ C00531 BC00531 VJ=50.00
MOVJ C00532 BC00532 VJ=50.00
'**********************
'W19B
'**********************
SFTON P0358
MOVL C00533 BC00533 V=500.0
MOVL C00534 BC00534 V=166.7 PL=0
SFTOF
ARCON
SFTON P0359
MOVL C00535 BC00535 V=10.8
ARCOF
SFTOF
MOVL C00536 BC00536 V=250.0
MOVJ C00537 BC00537 VJ=40.00
MOVJ C00538 BC00538 VJ=50.00
CALL JOB:MOVE_OUT_OF_TUNNEL
END
